# EPICS IOC start-up script: iocs/standaIOC/iocBoot/iocStanda/settings.iocsh
# prefix used for all PVs in this IOC
epicsEnvSet("PREFIX", "standa:")
